Yaskawa INFORM job: MULTI-BELOW.JBI

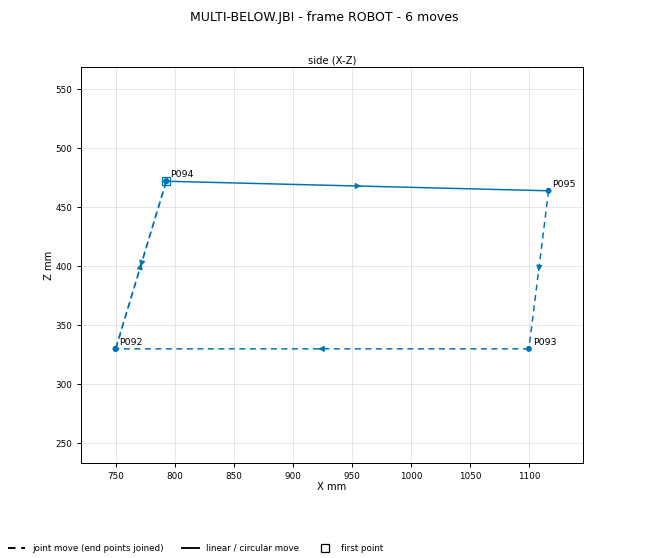
[picture p0: tool path of MULTI-BELOW.JBI in frame ROBOT, 6 of 6 moves have a stored position in this frame; points joined in program order, loops and branches not executed]
/JOB
//NAME MULTI-BELOW
///FOLDERNAME FOLDER001
//POS
///NPOS 2,0,0,4,0,0
///USER 15
///TOOL 1
///POSTYPE USER
///RECTAN
///RCONF 0,0,0,0,1,0,0,0,0,0,0,0,0,0,0,0,0,0,0,0,0,0,0,0
C00000=5.957,15.445,-75.515,0.0000,10.0000,0.0000
///LIMIT ON
C00001=5.866,-21.547,-75.511,180.0000,10.0000,0.0000
///POSTYPE ROBOT
///LIMIT OFF
///RCONF 0,0,0,0,0,0,0,0,0,0,0,0,0,0,0,0,0,0,0,0,0,0,0,0
P00092=750.003,161.812,330.004,0.1640,10.0066,0.1393
P00093=1100.002,161.807,330.008,0.1639,24.9999,0.1388
P00094=792.896,160.291,471.972,0.0813,10.0064,0.0684
P00095=1116.664,160.280,463.887,0.0787,10.0067,0.0664
//INST
///DATE 2025/05/21 10:37
///ATTR SC,RW,RJ
////FRAME USER 15
///GROUP1 RB1
///LVARS 20,20,20,0,0,0,0,0
NOP
MOVJ P094 VJ=15.00 PL=0
GETARG LB000 IARG#(1)
ADD B097 LB000
'=====
DOUT OT#(46) ON
TIMER T=0.50
JUMP LABEL: B099
*0
'ROOT
SFTOF
MACRO1 MJ#(2) ARGF2.4 ARGF1.5 ARGF0.0
MACRO1 MJ#(1) ARGF0.0 ARGF0.0 ARGF0.0 ARGF0.0 ARGF0.0 ARGF0.0
JUMP *LABEL
*1
'LAYER 1 - 1
SFTOF
MACRO1 MJ#(2) ARGF0.5 ARGF1.0 ARGF0.0
MACRO1 MJ#(1) ARGF0.0 ARGF-1.5 ARGF-3.0 ARGF5.0 ARGF0.0 ARGF0.0
JUMP *LABEL
*2
'LAYER 1 - 2
SFTOF
MACRO1 MJ#(2) ARGF0.5 ARGF1.0 ARGF0.0
MACRO1 MJ#(1) ARGF0.0 ARGF1.5 ARGF-3.0 ARGF-5.0 ARGF0.0 ARGF0.0
JUMP *LABEL
*3
'LAYER 2 - 1
SFTOF
MACRO1 MJ#(2) ARGF0.5 ARGF1.0 ARGF0.0
MACRO1 MJ#(1) ARGF0.0 ARGF3.0 ARGF-6.0 ARGF-7.0 ARGF0.0 ARGF0.0
JUMP *LABEL
*4
'LAYER 2 -2
SFTOF
MACRO1 MJ#(2) ARGF0.5 ARGF1.0 ARGF0.0
MACRO1 MJ#(1) ARGF0.0 ARGF-3.0 ARGF-6.0 ARGF7.0 ARGF0.0 ARGF0.0
JUMP *LABEL
*5
'LAYER 3 - 1
SFTOF
MACRO1 MJ#(2) ARGF0.5 ARGF1.0 ARGF0.0
MACRO1 MJ#(1) ARGF0.0 ARGF-6.0 ARGF-9.0 ARGF7.0 ARGF0.0 ARGF0.0
JUMP *LABEL
*6
'LAYER 3 - 2
SFTOF
MACRO1 MJ#(2) ARGF0.5 ARGF1.0 ARGF0.0
MACRO1 MJ#(1) ARGF0.0 ARGF0.0 ARGF-9.0 ARGF0.0 ARGF0.0 ARGF0.0
JUMP *LABEL
*7
'LAYER 3 - 3
SFTOF
MACRO1 MJ#(2) ARGF0.5 ARGF1.0 ARGF0.0
MACRO1 MJ#(1) ARGF0.0 ARGF6.0 ARGF-9.0 ARGF-7.0 ARGF0.0 ARGF0.0
JUMP *LABEL
*8
'LAYER 4 - 1
SFTOF
MACRO1 MJ#(2) ARGF0.5 ARGF1.0 ARGF0.0
MACRO1 MJ#(1) ARGF0.0 ARGF9.0 ARGF-13.0 ARGF-7.0 ARGF0.0 ARGF0.0
JUMP *LABEL
*9
'LAYER 4 - 2
SFTOF
MACRO1 MJ#(2) ARGF0.5 ARGF1.0 ARGF0.0
MACRO1 MJ#(1) ARGF0.0 ARGF3.0 ARGF-13.0 ARGF0.0 ARGF0.0 ARGF0.0
JUMP *LABEL
*10
'LAYER 4 - 3
SFTOF
MACRO1 MJ#(2) ARGF0.5 ARGF1.0 ARGF0.0
MACRO1 MJ#(1) ARGF0.0 ARGF-9.0 ARGF-13.0 ARGF7.0 ARGF0.0 ARGF0.0
JUMP *LABEL
*11
'LAYER 4 - 4
SFTOF
MACRO1 MJ#(2) ARGF0.5 ARGF1.0 ARGF0.0
MACRO1 MJ#(1) ARGF0.0 ARGF-3.0 ARGF-13.0 ARGF0.0 ARGF0.0 ARGF0.0
JUMP *LABEL
*12
'LAYER 5 - 1
SFTOF
MACRO1 MJ#(2) ARGF0.5 ARGF1.0 ARGF0.0
MACRO1 MJ#(1) ARGF0.0 ARGF-12.0 ARGF-18.0 ARGF7.0 ARGF0.0 ARGF0.0
JUMP *LABEL
*13
'LAYER 5 - 2
SFTOF
MACRO1 MJ#(2) ARGF0.5 ARGF1.0 ARGF0.0
MACRO1 MJ#(1) ARGF0.0 ARGF6.0 ARGF-18.0 ARGF0.0 ARGF0.0 ARGF0.0
JUMP *LABEL
*14
'LAYER 5 - 3
SFTOF
MACRO1 MJ#(2) ARGF0.5 ARGF1.0 ARGF0.0
MACRO1 MJ#(1) ARGF0.0 ARGF12.0 ARGF-18.0 ARGF-7.0 ARGF0.0 ARGF0.0
JUMP *LABEL
*15
'LAYER 5 - 4
SFTOF
MACRO1 MJ#(2) ARGF0.5 ARGF1.0 ARGF0.0
MACRO1 MJ#(1) ARGF0.0 ARGF-6.0 ARGF-18.0 ARGF0.0 ARGF0.0 ARGF0.0
JUMP *LABEL
*16
'LAYER 5 - 5
SFTOF
MACRO1 MJ#(2) ARGF0.5 ARGF1.0 ARGF0.0
MACRO1 MJ#(1) ARGF0.0 ARGF0.0 ARGF-18.0 ARGF0.0 ARGF0.0 ARGF0.0
JUMP *LABEL
*LABEL
REFP 1 C00000
REFP 2 C00001
MOVJ P092 VJ=15.00 PL=3
MOVJ P094 VJ=15.00 PL=0
ARCON
WVON AMP=D080 FREQ=D081 ANGL=D082
WVADJ STD=4.000 ST=1.000 END=2.000 LEN=400.000 ADJMD=0
MOVL P095 V=58.3 PL=0
WVOF
ARCOF
MOVJ P093 VJ=15.00 PL=3
MOVJ P092 VJ=15.00 PL=3
INC B099
SFTOF
JUMP LABEL: B099 IF B099<B097
SET B099 B097
END
